TYPE ST_EL1918 :
STRUCT
	//--------------------------------------------------------------------------------------------------------
	sTerminalName                                           :   STRING(200):= 'EL1918 | 8-Channel Safety Digital Input';
    //============================================================================================================================	
	// TERMINAL - EL1918 8-Channel Digital Input Terminal (Term 4)	
	iEL1918_Ch1                			AT %I*			: 	BOOL;	// EL1918 channel 1
	iEL1918_Ch2                   		AT %I*			: 	BOOL;	// EL1918 channel 2
	iEL1918_Ch3        					AT %I*	 		: 	BOOL;	// EL1918 channel 3
	iEL1918_Ch4   						AT %I*	 		: 	BOOL;	// EL1918 channel 4
	iEL1918_Ch5         				AT %I*	 		: 	BOOL;	// EL1918 channel 5 		     			
	iEL1918_Ch6 						AT %I*			: 	BOOL;	// EL1918 channel 6
	iEL1918_Ch7               			AT %I*          :   BOOL;   // EL1918 channel 7 
    iEL1918_Ch8          				AT %I*          :   BOOL;   // EL1918 channel 8
 		
	stTerminalInfo											: 	ST_Terminal_Info;

END_STRUCT
END_TYPE

(* stored: Version 1.1.0.1, ProductVersion 3.1.4026.18
   DUT ST_EL1918: Id {2006d025-ea4a-432a-beec-6893f1f5136f} *)
